PROGRAM PRG_HVCP3_48CB1
VAR
    // Function Block Instance
    fbDisconnector		: FB_DisconnectorControl;
	
	stDisconnectorIO	: ST_DisconnectorIO;
	
    
    // Başlangıç konfigürasyonu için flag
    bInitDone: BOOL := FALSE;	
END_VAR

IF NOT bInitDone THEN
	bInitDone := TRUE;
	RETURN;
END_IF

//*************************************************************************
// Ana Besleme Ayırıcısı
// +EP6-8CB1
//*************************************************************************
fbDisconnector(
    // Fiziksel Girişler
    bContactorOn_FB 	:= stDisconnectorIO.bContactorOn_FB,
    bContactorOff_FB 	:= stDisconnectorIO.bContactorOff_FB,
    bLimitOn 			:= stDisconnectorIO.bLimitOn,
    bLimitOff 			:= stDisconnectorIO.bLimitOff,
    bThermalFault 		:= stDisconnectorIO.bThermalFault,
    bEarthSwitchOn 		:= stDisconnectorIO.bEarthSwitchOn,
    bEarthSwitchOff 	:= stDisconnectorIO.bEarthSwitchOff,
    bPLCControl 		:= stDisconnectorIO.bPLCControl,
    
    // Güvenlik Girişleri
    bSafetyLoop 		:= GVL_Alarm.bSafetyLoop,
    bInterlock 			:= FALSE,
    
    // Sistem Girişleri
    bMasterReset 		:= GVL_Alarm.bMasterReset,
    
    // HMI Bağlantısı
    stHMI 				:= GVL_HVCP3.st48CB1HMI,
    
    // Fiziksel Çıkışlar
    bContactorOn_Out 	=> stDisconnectorIO.bContactorOn_Out,
    bContactorOff_Out 	=> stDisconnectorIO.bContactorOff_Out
);

METHOD M_Init : BOOL
VAR_INPUT
END_VAR

GVL_HVCP3.st16CB1HMI.stConfig.bEarthSwitchExists := FALSE;
GVL_HVCP3.st16CB1HMI.stConfig.bGrounded := FALSE;
GVL_HVCP3.st16CB1HMI.stConfig.bInterlockEnable := TRUE;
GVL_HVCP3.st16CB1HMI.stConfig.dwOperationLimit := 10000;
GVL_HVCP3.st16CB1HMI.stConfig.nPhaseCount := 3;
GVL_HVCP3.st16CB1HMI.stConfig.rRatedCurrent := 1000.0;
GVL_HVCP3.st16CB1HMI.stConfig.rRatedVoltage := 36000.0;
GVL_HVCP3.st16CB1HMI.stConfig.sProductCode := '';
GVL_HVCP3.st16CB1HMI.stConfig.sProjectCode := '+EP9-48CB1';
GVL_HVCP3.st16CB1HMI.stConfig.tContactorDelay := T#500MS;
GVL_HVCP3.st16CB1HMI.stConfig.tMotionTimeout := T#50S;
END_METHOD

END_PROGRAM

(* stored: Version 1.1.0.1, ProductVersion 3.1.4024.15
   POU PRG_HVCP3_48CB1: Id {c109f43b-25d1-408a-ac2e-e1ea8e66f55b}, SpecialFunc None
   Method M_Init: Id {a00478c3-a8b7-4f1a-8500-5046a8ba48d6} *)
